% RSLogix 500 project Hanout 5 Motor Problem AJ.RSS, saved by version 10.00.00.00 %
PROJECT "ML06A"    % processor: Bul.1763 MicroLogix 1100 Series B %

PROGRAM FILES
  LAD 2   6 rungs

DATA FILES
  O0 OUTPUT  4 elements
  I1 INPUT  6 elements
  S2 STATUS  66 elements
  B3 BINARY  1 elements
  T4 TIMER  1 elements
  C5 COUNTER  1 elements
  R6 CONTROL  1 elements
  N7 INTEGER  1 elements
  F8 FLOAT  1 elements

LADDER 2
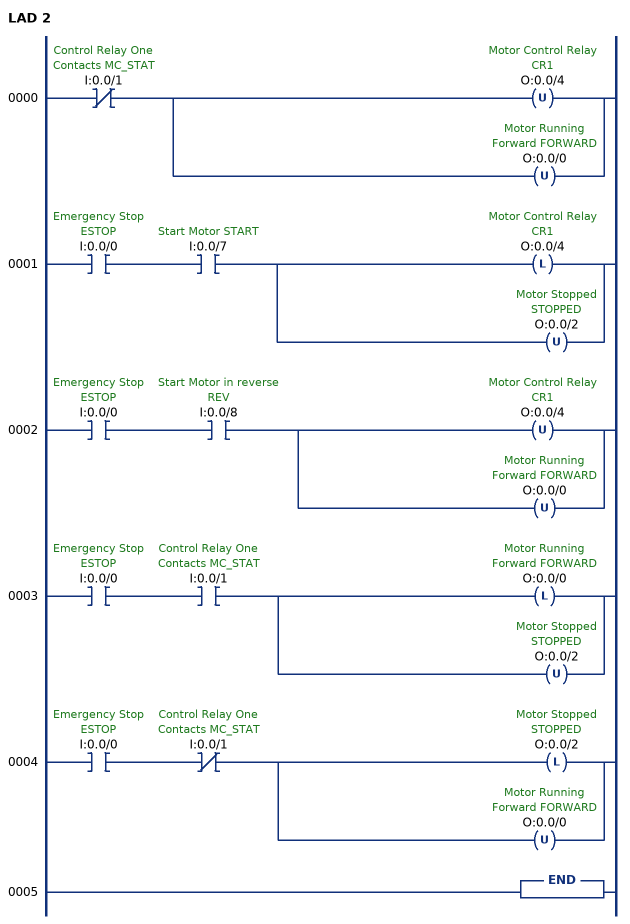
% Rung: 0 %
SOR XIO I:0.0/1 BST OTU O:0.0/4 NXB OTU O:0.0/0 BND EOR
%   I:0.0/1  MC_STAT  "Control Relay One Contacts" %
%   O:0.0/4  CR1  "Motor Control Relay" %
%   O:0.0/0  FORWARD  "Motor Running Forward" %
% Rung: 1 %
SOR XIC I:0.0/0 XIC I:0.0/7 BST OTL O:0.0/4 NXB OTU O:0.0/2 BND EOR
%   I:0.0/0  ESTOP  "Emergency Stop" %
%   I:0.0/7  START  "Start Motor" %
%   O:0.0/4  CR1  "Motor Control Relay" %
%   O:0.0/2  STOPPED  "Motor Stopped" %
% Rung: 2 %
SOR XIC I:0.0/0 XIC I:0.0/8 BST OTU O:0.0/4 NXB OTU O:0.0/0 BND EOR
%   I:0.0/0  ESTOP  "Emergency Stop" %
%   I:0.0/8  REV  "Start Motor in reverse" %
%   O:0.0/4  CR1  "Motor Control Relay" %
%   O:0.0/0  FORWARD  "Motor Running Forward" %
% Rung: 3 %
SOR XIC I:0.0/0 XIC I:0.0/1 BST OTL O:0.0/0 NXB OTU O:0.0/2 BND EOR
%   I:0.0/0  ESTOP  "Emergency Stop" %
%   I:0.0/1  MC_STAT  "Control Relay One Contacts" %
%   O:0.0/0  FORWARD  "Motor Running Forward" %
%   O:0.0/2  STOPPED  "Motor Stopped" %
% Rung: 4 %
SOR XIC I:0.0/0 XIO I:0.0/1 BST OTL O:0.0/2 NXB OTU O:0.0/0 BND EOR
%   I:0.0/0  ESTOP  "Emergency Stop" %
%   I:0.0/1  MC_STAT  "Control Relay One Contacts" %
%   O:0.0/2  STOPPED  "Motor Stopped" %
%   O:0.0/0  FORWARD  "Motor Running Forward" %
% Rung: 5 %
SOR END EOR

OTHER DOCUMENTED ADDRESSES
  B3:0/0  ESTOP_STOP_BIT  "Estop/stop info bit"
  B3:0/1  FWD_BIT  "Forward direction bit"
  B3:0/2  REV_BIT  "Reverse direction bit"
  B3:0/3  LAST_FWD  "Motor Last In Forward"
  B3:0/4  LAST_REV  "Motor Last In Reverse"
  I:0.0/2  DIR_STAT  "Control Relay Two Contacts"
  I:0.0/3  DIR_F  "Forward direction 3PSS"
  I:0.0/4  DIR_R  "Reverse direction 3PSS"
  I:0.0/5  RUN_JOG  "Run/Jog Mode"
  I:0.0/6  STOP  "Stop Motor"
  MOV  
  O:0.0/1  CHANGING  "Motor Direction Change"
  O:0.0/3  REVERSE  "Motor Running Reverse"
  O:0.0/5  CR2  "Direction Control Relay"
  PB1  "Start Motor"
  T4:0  TIME_ON_DELAY  "Keeps motor stopped when switching to forward/reverse"
  T4:0/DN  T4
  T4:0/TT  MOTOR_CHANGE_TIMER  "Timer for motor change"

DATA TABLE (non-zero values as saved)
DATA T4
% .PRE .ACC %
% T4:0 % 16 0
DATA C5
% .PRE .ACC %
% C5:0 % 16 3
